// TIA Portal V16 export
// export: Created 2021-05-25T16:14:32.3672726Z, ExportSetting WithDefaults, DisplayName Totally Integrated Automation Portal, DisplayVersion V16, DisplayName TIA Portal Version Control Interface, DisplayVersion V16, DisplayName TIA Portal Openness, DisplayVersion V16, DisplayName STEP 7 Professional, DisplayVersion V16, DisplayName STEP 7 Safety, DisplayVersion V16, DisplayName WinCC Unified SCADA Engineering System, DisplayVersion V16
ORGANIZATION_BLOCK "Main"   // OB1, LAD, ProgramCycle
TITLE = "Main Program Sweep (Cycle)"
{ S7_Optimized_Access := 'TRUE' }
VERSION : 0.1
// stored: AutoNumber true, IsIECCheckEnabled false, SetENOAutomatically false
   VAR_INPUT
      Initial_Call : Bool;   // Initial call of this OB
      Remanence : Bool;   // =True, if remanent data are available
   END_VAR
   VAR_TEMP
      OB1_SCAN_1 : Byte;   // 1 (Cold restart scan 1 of OB 1), 3 (Scan 2-n of OB 1)
      OB1_PRIORITY : Byte;   // Priority of OB Execution
      OB1_OB_NUMBR : Byte;   // 1 (Organization block 1, OB1)
      OB1_RESERVED_1 : Byte;   // Reserved for system
      OB1_RESERVED_2 : Byte;   // Reserved for system
      OB1_EV_CLASS : Byte;   // Bits 0-3 = 1 (Coming event), Bits 4-7 = 1 (Event class 1)
      OB1_PREV_CYCLE : Int;   // Cycle time of previous OB1 scan (milliseconds)
      OB1_MIN_CYCLE : Int;   // Minimum cycle time of OB1 (milliseconds)
      OB1_MAX_CYCLE : Int;   // Maximum cycle time of OB1 (milliseconds)
      OB1_DATE_TIME : DTL;   // Date and time OB1 started
   END_VAR
BEGIN

REGION Network 1
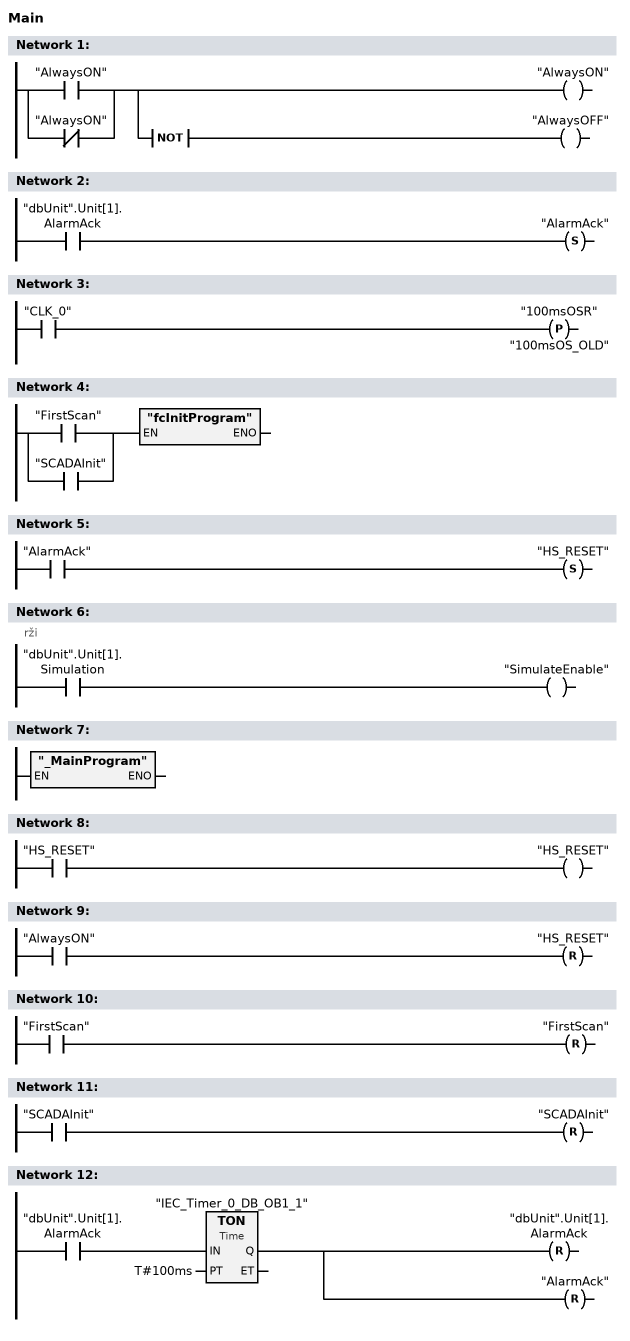
   RUNG wire#powerrail
      Contact( "AlwaysON" )
      wire#w1
      Coil( "AlwaysON" )
   END_RUNG
   RUNG wire#powerrail
      I_Contact( "AlwaysON" )
   END_RUNG wire#w1
   RUNG wire#w1
      Not()
      Coil( "AlwaysOFF" )
   END_RUNG
   // the same network as SCL:
   "AlwaysON" := "AlwaysON" OR NOT "AlwaysON";
   "AlwaysOFF" := NOT "AlwaysON";
END_REGION

REGION Network 2
   RUNG wire#powerrail
      Contact( "dbUnit".Unit[1].AlarmAck )
      S_Coil( "AlarmAck" )
   END_RUNG
   // the same network as SCL:
   IF "dbUnit".Unit[1].AlarmAck THEN "AlarmAck" := TRUE; END_IF;
END_REGION

REGION Network 3
   "100msOSR" := "CLK_0" AND NOT "100msOS_OLD";   // rising edge
   "100msOS_OLD" := "CLK_0";
END_REGION

REGION Network 4
   RUNG wire#powerrail
      Contact( "FirstScan" )
      wire#w1
      "fcInitProgram"()
   END_RUNG
   RUNG wire#powerrail
      Contact( "SCADAInit" )
   END_RUNG wire#w1
   // the same network as SCL:
   IF "FirstScan" OR "SCADAInit" THEN "fcInitProgram"(); END_IF;
END_REGION

REGION Network 5
   RUNG wire#powerrail
      Contact( "AlarmAck" )
      S_Coil( "HS_RESET" )
   END_RUNG
   // the same network as SCL:
   IF "AlarmAck" THEN "HS_RESET" := TRUE; END_IF;
END_REGION

REGION Network 6
   // rži
   RUNG wire#powerrail
      Contact( "dbUnit".Unit[1].Simulation )
      Coil( "SimulateEnable" )
   END_RUNG
   // the same network as SCL:
   "SimulateEnable" := "dbUnit".Unit[1].Simulation;
END_REGION

REGION Network 7
   RUNG wire#powerrail
      "_MainProgram"()
   END_RUNG
   // the same network as SCL:
   "_MainProgram"();
END_REGION

REGION Network 8
   RUNG wire#powerrail
      Contact( "HS_RESET" )
      Coil( "HS_RESET" )
   END_RUNG
   // the same network as SCL:
   "HS_RESET" := "HS_RESET";
END_REGION

REGION Network 9
   RUNG wire#powerrail
      Contact( "AlwaysON" )
      R_Coil( "HS_RESET" )
   END_RUNG
   // the same network as SCL:
   IF "AlwaysON" THEN "HS_RESET" := FALSE; END_IF;
END_REGION

REGION Network 10
   RUNG wire#powerrail
      Contact( "FirstScan" )
      R_Coil( "FirstScan" )
   END_RUNG
   // the same network as SCL:
   IF "FirstScan" THEN "FirstScan" := FALSE; END_IF;
END_REGION

REGION Network 11
   RUNG wire#powerrail
      Contact( "SCADAInit" )
      R_Coil( "SCADAInit" )
   END_RUNG
   // the same network as SCL:
   IF "SCADAInit" THEN "SCADAInit" := FALSE; END_IF;
END_REGION

REGION Network 12
   RUNG wire#powerrail
      Contact( "dbUnit".Unit[1].AlarmAck )
      { S7_Templates := "time_type := Time" } "IEC_Timer_0_DB_OB1_1".TON(pt := T#100ms, et =>)
      wire#w1
      R_Coil( "dbUnit".Unit[1].AlarmAck )
   END_RUNG
   RUNG wire#w1
      R_Coil( "AlarmAck" )
   END_RUNG
   // the same network as SCL:
   "IEC_Timer_0_DB_OB1_1".TON(IN := "dbUnit".Unit[1].AlarmAck, PT := T#100ms);
   IF "IEC_Timer_0_DB_OB1_1".Q THEN
       "dbUnit".Unit[1].AlarmAck := FALSE;
       "AlarmAck" := FALSE;
   END_IF;
END_REGION
END_ORGANIZATION_BLOCK
